(* PLC project SafeLOGIC-1, BrAutomation SafeDESIGNER  4.3.4.4 *)
(* stored: companyURL http://www.br-automation.com, creationDateTime Mon Dec 02 13:04:35 2019 *)

PROGRAM Main

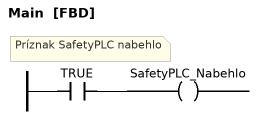
(* FBD diagram, written out as Structured Text *)
(* Príznak SafetyPLC nabehlo *)
SafetyPLC_Nabehlo := TRUE;
END_PROGRAM
